(* IEC 61131-3 sources: Caravan/Archiv/12-04-19/Stations/MachineControl/MachineControl/Class/InputMyIO, 1 file *)

(* ---- InputMyIO.st ---- *)
(*!
<Class
	Name               = "InputMyIO"
	Revision           = "0.0"
	RealtimeTask       = "false"
	CyclicTask         = "false"
	DefCyclictime      = "10 ms"
	BackgroundTask     = "false"
	Sigmatek           = "false"
	OSInterface        = "false"
	HighPriority       = "false"
	Automatic          = "false"
	UpdateMode         = "Prescan"
	SharedCommandTable = "true"
	Objectsize         = "(308,120)">
	<Channels>
		<Server Name="sXDir" Visualized="true" Initialize="false" WriteProtected="false" Retentive="false"/>
		<Server Name="sYDir" Visualized="true" Initialize="false" WriteProtected="false" Retentive="false"/>
		<Client Name="oc_Grafix" Required="false" Internal="false"/>
	</Channels>
	<Network Name="InputMyIO">
		<!-- List of Components in this network -->
		<Components>
			<Object
				Name       = "_base"
				Class      = "_MyIO"
				Position   = "(218,120)"
				Visualized = "true"
				Remotely   = "true">
				<Channels>
					<Server Name="Refresh"/>
					<Server Name="Server0"/>
					<Client Name="Graphic"/>
					<Client Name="Lse"/>
				</Channels>
			</Object>
		</Components>
		<Comments>
		</Comments>
		<!-- List of Connections in this network -->
		<Connections>
			<Connection Source="this.Server0" Destination="_base.Server0" Vertices="(690,210),(518,210),"/>
			<Connection Source="this.Refresh" Destination="_base.Refresh" Vertices="(690,270),(518,270),"/>
			<Connection Source="_base.Lse" Destination="this.Lse" Vertices="(218,210),(38,210),"/>
		</Connections>
		<!-- Headerfiles -->
		<Options>
		</Options>
	</Network>
</Class>
*)
#pragma using _MyIO

InputMyIO : CLASS
: _MyIO
  //Servers:
	sXDir 	: SvrCh_DINT;
	sYDir 	: SvrCh_DINT;
  //Clients:
	oc_Grafix 	: CltChCmd__Grafix;
  //Variables:
		bMyFocus 	: BOOL;
  //Functions:
				//! <Function Comment="this method will be called once when the focus will be given to this object" Name="GetFocus"/>
	FUNCTION __CDECL VIRTUAL GLOBAL GetFocus
		VAR_INPUT
			pio 	: ^_IO;			//! <Variable Comment="pointer to _IO information" Name="GetFocus.pio"/>
		END_VAR
		VAR_OUTPUT
			retcode (EAX) 	: _DOIT;			//! <Variable Comment="return _IFAILED if you dont want to get the focus on the other hand _IDLE" Name="GetFocus.retcode"/>
		END_VAR;
				//! <Function Comment="this method is called once when the focus is taken from object" Name="KillFocus"/>
	FUNCTION __CDECL VIRTUAL GLOBAL KillFocus
		VAR_INPUT
			pio 	: ^_IO;			//! <Variable Comment="pointer to _IO information" Name="KillFocus.pio"/>
		END_VAR
		VAR_OUTPUT
			retcode (EAX) 	: _DOIT;			//! <Variable Comment="return always _IDLE because you can&apos;t prevent action" Name="KillFocus.retcode"/>
		END_VAR;
				//! <Function Comment="this method is called everytime when the input is active and a event occured" Name="GetEvent"/>
	FUNCTION __CDECL VIRTUAL GLOBAL GetEvent
		VAR_INPUT
			ped 	: ^_EDITOR;			//! <Variable Comment="pointer to _EDITOR information" Name="GetEvent.ped"/>
			pe 	: ^_EVENT;			//! <Variable Comment="pointer to _EVENT information" Name="GetEvent.pe"/>
		END_VAR
		VAR_OUTPUT
			retcode (EAX) 	: _DOIT;			//! <Variable Comment="for the returnstatement there are 3 different possibilities&#13;&#10;  _IDLE ..... the system should goon like it is (system goes on)&#13;&#10;  _IDIDIT ... i did it (system is ready)&#13;&#10;  _IFAILED .. i tried to do my best, but i failed (system is ready)&#13;&#10;" Name="GetEvent.retcode"/>
		END_VAR;
				//! <Function Comment="this method is called everytime when system wants to redraw the io" Name="Draw"/>
	FUNCTION __CDECL VIRTUAL GLOBAL Draw
		VAR_INPUT
			pio 	: ^_IO;			//! <Variable Comment="pointer to _IO information" Name="Draw.pio"/>
			pr 	: ^_RESULT;			//! <Variable Comment="pointer to _RESULT information" Name="Draw.pr"/>
			pv 	: ^_VARIABLE;			//! <Variable Comment="pointer to io _VARIABLE information" Name="Draw.pv"/>
			input 	: BOOL;			//! <Variable Comment="TRUE it&apos;s an input&#13;&#10;FALSE it&apos;s an output" Name="Draw.input"/>
		END_VAR
		VAR_OUTPUT
			retcode (EAX) 	: _DOIT;			//! <Variable Comment="for the returnstatement there are 3 different possibilities&#13;&#10;  _IDLE ..... the system should goon like it is (system goes on)&#13;&#10;  _IDIDIT ... i did it (system is ready)&#13;&#10;  _IFAILED .. i tried to do my best, but i failed (system is re" Name="Draw.retcode"/>
		END_VAR;
				//! <Function Comment="this method is called everytime when system wants to get data for defined io.&#13;&#10;&#13;&#10;pr ........ &#13;&#10;pio ....... pointer to io information&#13;&#10;pv ........ pointer to io variableinformation&#13;&#10;input ..... TRUE it&apos;s an input / FALSE it&apos;s an output&#13;&#10;&#13;&#10;for the returnstatement there are 3 different possibilities&#13;&#10;_IDLE ..... the system should goon like it is (system goes on)&#13;&#10;_IDIDIT ... i did it (system is ready)&#13;&#10;_IFAILED .. i tried to do my best, but i failed (system is ready)&#13;&#10;&#13;&#10;if you want to do it let&apos;s return _IDIDIT and initialize the  structure _RESULT&#13;&#10;" Name="GetData"/>
	FUNCTION __CDECL VIRTUAL GLOBAL GetData
		VAR_INPUT
			pr 	: ^_RESULT;			//! <Variable Comment="pointer to _RESULT information" Name="GetData.pr"/>
			pio 	: ^_IO;			//! <Variable Comment="pointer to _IO information" Name="GetData.pio"/>
			pv 	: ^_VARIABLE;			//! <Variable Comment="pointer to _VARIABLE information given by LSE" Name="GetData.pv"/>
			input 	: BOOL;			//! <Variable Comment="TRUE it&apos;s an input&#13;&#10;FALSE it&apos;s an output" Name="GetData.input"/>
		END_VAR
		VAR_OUTPUT
			retcode (EAX) 	: _DOIT;			//! <Variable Comment="for the returnstatement there are 3 different possibilities&#13;&#10;  _IDLE ..... the system should goon like it is (system goes on)&#13;&#10;  _IDIDIT ... i did it (system is ready)&#13;&#10;  _IFAILED .. i tried to do my best, but i failed (system is ready)" Name="GetData.retcode"/>
		END_VAR;
  //Tables:
	FUNCTION @STD
		VAR_OUTPUT
			ret_code	: CONFSTATES;
		END_VAR;
	FUNCTION GLOBAL TAB @CT_;
END_CLASS;

#pragma usingLtd _Grafix

FUNCTION __CDECL VIRTUAL GLOBAL InputMyIO::GetData
	VAR_INPUT
		pr 	: ^_RESULT;
		pio 	: ^_IO;
		pv 	: ^_VARIABLE;
		input 	: BOOL;
	END_VAR
	VAR_OUTPUT
		retcode (EAX) 	: _DOIT;
	END_VAR

  _MyIO::GetData(pr:=pr, pio:=pio, pv:=pv, input:=input);
  // pr : pointer auf Serverdaten
  pr^.value := TO_DINT((TO_UDINT(sXDir) rol 1) xor (TO_UDINT(sYDir)));
  retcode := _IDIDIT;

END_FUNCTION

FUNCTION __CDECL VIRTUAL GLOBAL InputMyIO::GetEvent
	VAR_INPUT
		ped 	: ^_EDITOR;
		pe 	: ^_EVENT;
	END_VAR
	VAR_OUTPUT
		retcode (EAX) 	: _DOIT;
	END_VAR

  _MyIO::GetEvent(ped:=ped, pe:=pe);

  retcode := _IDLE;

  if pe^.ftype = _EVENT_HIDMOVE then

    if (pe^.dot.x >= ped^.input.io.space.xy1.x) &
       (pe^.dot.x <= ped^.input.io.space.xy2.x) &
       (pe^.dot.y >= ped^.input.io.space.xy1.y) &
       (pe^.dot.y <= ped^.input.io.space.xy2.y) then

       sXDir := pe^.dot.x - ped^.input.io.space.xy1.x;
       sYDir := ped^.input.io.space.xy2.y - pe^.dot.y;

       retcode := _IDIDIT;

    end_if;
  end_if;

END_FUNCTION

FUNCTION __CDECL VIRTUAL GLOBAL InputMyIO::Draw
	VAR_INPUT
		pio 	: ^_IO;
		pr 	: ^_RESULT;
		pv 	: ^_VARIABLE;
		input 	: BOOL;
	END_VAR
	VAR_OUTPUT
		retcode (EAX) 	: _DOIT;
	END_VAR
  VAR
  	act   : _NEWSCREEN;
    x     : _KOORD;
    y     : _KOORD;
    color : _COLOR;
  END_VAR

  _MyIO::Draw(pio:=pio, pr:=pr, pv:=pv, input:=input);

  x := pio^.space.xy1.x + TO_INT(sXDir);
  y := pio^.space.xy2.y - TO_INT(sYDir);

  if (bMyFocus = TRUE) then
    color := GetEditColorBack(x0:=_EDITACTIVE);
  else
    color := pio^.coltxt;
  end_if;

  push_screen(p0:=#act);

  oc_Grafix.PutImage(image:=#pio^.image,
                     x0:=DEFKOORD,
                     y0:=DEFKOORD);

  oc_Grafix.Rectangle(x0:= pio^.space.xy1.x,
                      y0:= pio^.space.xy1.y,
                      x1:= pio^.space.xy2.x,
                      y1:= pio^.space.xy2.y,
                      attrib:= pio^.attrib,
                      color:= pio^.colframe);

  oc_Grafix.Line(x0:=pio^.space.xy1.x,
                 y0:=y,
                 x1:=pio^.space.xy2.x,
                 y1:=y,
                 attrib:=pio^.attrib,
                 color:=color);

  oc_Grafix.Line(x0:=x,
                 y0:=pio^.space.xy1.y,
                 x1:=x,
                 y1:=pio^.space.xy2.y,
                 attrib:=pio^.attrib,
                 color:=color);

  pop_screen(p0:=#act);
  copy_screen(p0:=#act, p1:=#pio^.space);

  retcode := _IDIDIT;

  END_FUNCTION

FUNCTION __CDECL VIRTUAL GLOBAL InputMyIO::GetFocus
	VAR_INPUT
		pio 	: ^_IO;
	END_VAR
	VAR_OUTPUT
		retcode (EAX) 	: _DOIT;
	END_VAR

  _MyIO::GetFocus(pio:=pio);

  bMyFocus := TRUE;
  retcode := _IDLE;

END_FUNCTION

FUNCTION __CDECL VIRTUAL GLOBAL InputMyIO::KillFocus
	VAR_INPUT
		pio 	: ^_IO;
	END_VAR
	VAR_OUTPUT
		retcode (EAX) 	: _DOIT;
	END_VAR

  _MyIO::KillFocus(pio:=pio);

  bMyFocus := FALSE;
  retcode := _IDLE;

END_FUNCTION
